// Type alias for a file path wide string.
// [note] Change the maximum length of the path string in `PARAM_Constants.PATH_LENGTH`
TYPE T_WPath : WSTRING(PARAM_Constants.PATH_LENGTH); END_TYPE

(* stored: Version 1.1.0.1
   DUT T_WPath: Id {b4fbd076-e3bf-0136-08c9-6131a31ceb0d} *)
